% RSLogix 500 project timer question 3.RSS, saved by version 8.30.00.15 %
PROJECT "UNTITLED"    % processor: MicroLogix 1000 %

PROGRAM FILES
  LAD 2 "MAIN_PROG"  8 rungs
  LAD 3 "USER_FAULT"  1 rungs
  LAD 4 "HSC_INT"  1 rungs
  LAD 5 "STI_INT"  1 rungs
  LAD 6, 7, 8, 9, 10, 11, 12, 13, 14, 15, 16: only END

DATA FILES
  O0 OUTPUT  1 elements
  I1 INPUT  2 elements
  S2 STATUS  33 elements
  B3 BINARY  32 elements
  T4 TIMER  40 elements
  C5 COUNTER  32 elements
  R6 CONTROL  16 elements
  N7 INTEGER  105 elements

LADDER 2 "MAIN_PROG"
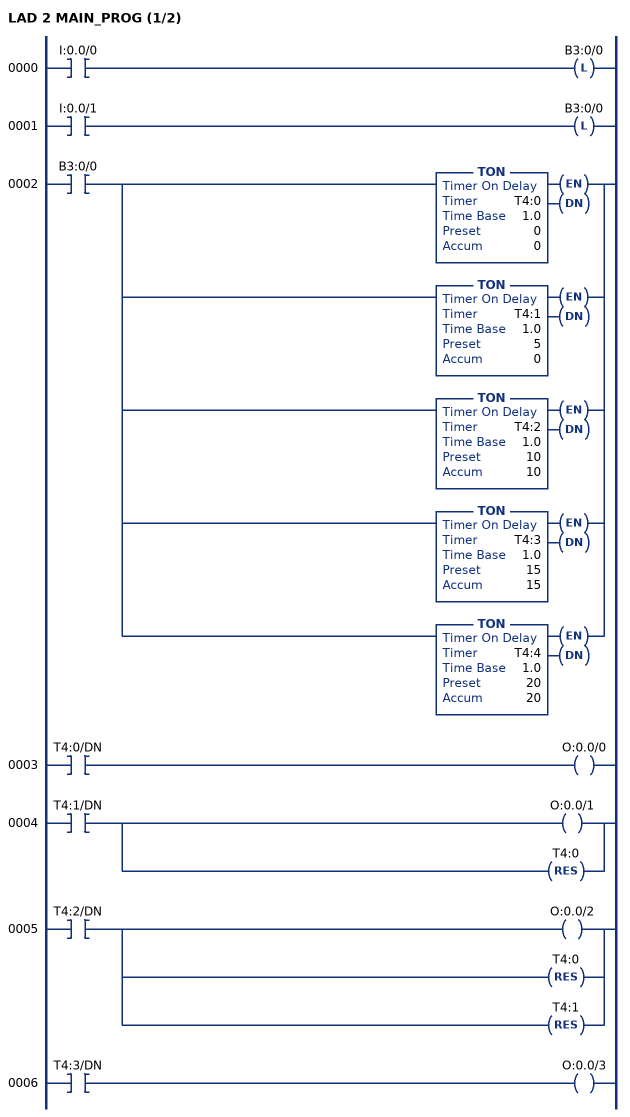
% Rung: 0 %
SOR XIC I:0.0/0 OTL B3:0/0 EOR
% Rung: 1 %
SOR XIC I:0.0/1 OTL B3:0/0 EOR
% Rung: 2 %
SOR XIC B3:0/0 BST BST BST BST TON T4:0 1.0 0 0 NXB TON T4:1 1.0 5 0 BND NXB TON T4:2 1.0 10 10 BND NXB TON T4:3 1.0 15 15 BND NXB TON T4:4 1.0 20 20 BND EOR
% Rung: 3 %
SOR XIC T4:0/DN OTE O:0.0/0 EOR
% Rung: 4 %
SOR XIC T4:1/DN BST OTE O:0.0/1 NXB RES T4:0 BND EOR
% Rung: 5 %
SOR XIC T4:2/DN BST BST OTE O:0.0/2 NXB RES T4:0 BND NXB RES T4:1 BND EOR
% Rung: 6 %
SOR XIC T4:3/DN OTE O:0.0/3 EOR

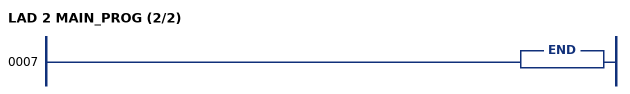
% Rung: 7 %
SOR END EOR

DATA TABLE (non-zero values as saved)
DATA B3
% B3:0 % 0X0001 0X0000 0X0000 0X0000 0X0000 0X0000 0X0000 0X0000 0X0000 0X0000
DATA T4
% .PRE .ACC %
% T4:1 % 5 0
% T4:2 % 10 10
% T4:3 % 15 15
% T4:4 % 20 20
